// TIA Portal V17 export
// export: Created 2022-07-20T06:59:37.911436Z, ExportSetting WithDefaults, DisplayName Totally Integrated Automation Portal, DisplayVersion V17, DisplayName TIA Portal Openness, DisplayVersion V17, DisplayName TIA Portal Version Control Interface, DisplayVersion V17, DisplayName SINAMICS Startdrive Advanced, DisplayVersion V17, DisplayName SINAMICS Startdrive G130, G150, S120, S150, SINAMICS MV, S210, DisplayVersion V17, DisplayName SINAMICS Startdrive G110M, G120, G120C, G120D, G120P, G115D, DisplayVersion V17, DisplayName STEP 7 Professional, DisplayVersion V17, DisplayName STEP 7 Safety, DisplayVersion V17, DisplayName WinCC Advanced, DisplayVersion V17
FUNCTION_BLOCK "FB10010_BoolToWordAT"   // FB10010, LAD
TITLE = FB10010_BoolToWordAT
{ S7_Optimized_Access := 'TRUE' }
AUTHOR : Jonathan
FAMILY : 1001x_CONVERT
VERSION : 1.0
// Release note : 
// 1.0 - Feature developped
// stored: AutoNumber false, IsIECCheckEnabled false, IsRetainMemResEnabled false, MemoryReserve 100, SetENOAutomatically false, UDAEnableTagReadback false
   VAR_INPUT
      bool0 { ExternalAccessible := 'False'; ExternalVisible := 'False'; ExternalWritable := 'False'} : Bool;
      bool1 { ExternalAccessible := 'False'; ExternalVisible := 'False'; ExternalWritable := 'False'} : Bool;
      bool2 { ExternalAccessible := 'False'; ExternalVisible := 'False'; ExternalWritable := 'False'} : Bool;
      bool3 { ExternalAccessible := 'False'; ExternalVisible := 'False'; ExternalWritable := 'False'} : Bool;
      bool4 { ExternalAccessible := 'False'; ExternalVisible := 'False'; ExternalWritable := 'False'} : Bool;
      bool5 { ExternalAccessible := 'False'; ExternalVisible := 'False'; ExternalWritable := 'False'} : Bool;
      bool6 { ExternalAccessible := 'False'; ExternalVisible := 'False'; ExternalWritable := 'False'} : Bool;
      bool7 { ExternalAccessible := 'False'; ExternalVisible := 'False'; ExternalWritable := 'False'} : Bool;
      bool8 { ExternalAccessible := 'False'; ExternalVisible := 'False'; ExternalWritable := 'False'} : Bool;
      bool9 { ExternalAccessible := 'False'; ExternalVisible := 'False'; ExternalWritable := 'False'} : Bool;
      bool10 { ExternalAccessible := 'False'; ExternalVisible := 'False'; ExternalWritable := 'False'} : Bool;
      bool11 { ExternalAccessible := 'False'; ExternalVisible := 'False'; ExternalWritable := 'False'} : Bool;
      bool12 { ExternalAccessible := 'False'; ExternalVisible := 'False'; ExternalWritable := 'False'} : Bool;
      bool13 { ExternalAccessible := 'False'; ExternalVisible := 'False'; ExternalWritable := 'False'} : Bool;
      bool14 { ExternalAccessible := 'False'; ExternalVisible := 'False'; ExternalWritable := 'False'} : Bool;
      bool15 { ExternalAccessible := 'False'; ExternalVisible := 'False'; ExternalWritable := 'False'} : Bool;
   END_VAR
   VAR_OUTPUT
      OutWord { ExternalAccessible := 'False'; ExternalVisible := 'False'; ExternalWritable := 'False'} : Word;
   END_VAR
   VAR DB_SPECIFIC
      statOutWord : Word;
   END_VAR
   VAR
      statbools AT statOutWord : Array[0..15] of Bool;
   END_VAR
BEGIN

REGION Network 1
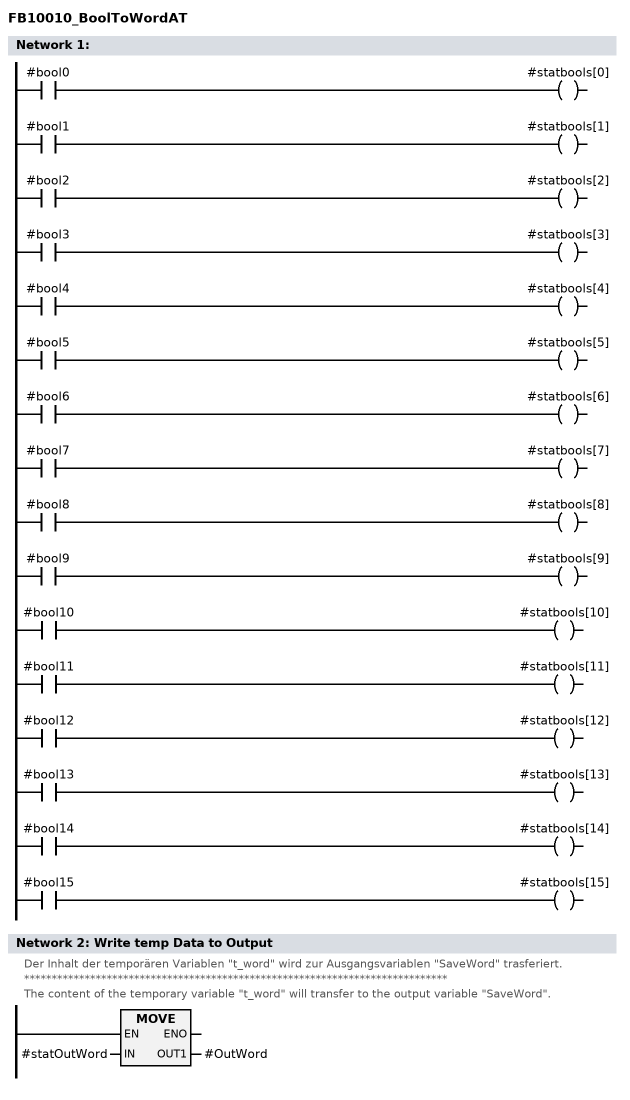
   RUNG wire#powerrail
      Contact( #bool0 )
      Coil( #statbools[0] )
   END_RUNG
   RUNG wire#powerrail
      Contact( #bool1 )
      Coil( #statbools[1] )
   END_RUNG
   RUNG wire#powerrail
      Contact( #bool2 )
      Coil( #statbools[2] )
   END_RUNG
   RUNG wire#powerrail
      Contact( #bool3 )
      Coil( #statbools[3] )
   END_RUNG
   RUNG wire#powerrail
      Contact( #bool4 )
      Coil( #statbools[4] )
   END_RUNG
   RUNG wire#powerrail
      Contact( #bool5 )
      Coil( #statbools[5] )
   END_RUNG
   RUNG wire#powerrail
      Contact( #bool6 )
      Coil( #statbools[6] )
   END_RUNG
   RUNG wire#powerrail
      Contact( #bool7 )
      Coil( #statbools[7] )
   END_RUNG
   RUNG wire#powerrail
      Contact( #bool8 )
      Coil( #statbools[8] )
   END_RUNG
   RUNG wire#powerrail
      Contact( #bool9 )
      Coil( #statbools[9] )
   END_RUNG
   RUNG wire#powerrail
      Contact( #bool10 )
      Coil( #statbools[10] )
   END_RUNG
   RUNG wire#powerrail
      Contact( #bool11 )
      Coil( #statbools[11] )
   END_RUNG
   RUNG wire#powerrail
      Contact( #bool12 )
      Coil( #statbools[12] )
   END_RUNG
   RUNG wire#powerrail
      Contact( #bool13 )
      Coil( #statbools[13] )
   END_RUNG
   RUNG wire#powerrail
      Contact( #bool14 )
      Coil( #statbools[14] )
   END_RUNG
   RUNG wire#powerrail
      Contact( #bool15 )
      Coil( #statbools[15] )
   END_RUNG
   // the same network as SCL:
   #statbools[0] := #bool0;
   #statbools[1] := #bool1;
   #statbools[2] := #bool2;
   #statbools[3] := #bool3;
   #statbools[4] := #bool4;
   #statbools[5] := #bool5;
   #statbools[6] := #bool6;
   #statbools[7] := #bool7;
   #statbools[8] := #bool8;
   #statbools[9] := #bool9;
   #statbools[10] := #bool10;
   #statbools[11] := #bool11;
   #statbools[12] := #bool12;
   #statbools[13] := #bool13;
   #statbools[14] := #bool14;
   #statbools[15] := #bool15;
END_REGION

REGION Network 2: Write temp Data to Output
   // Der Inhalt der temporären Variablen "t_word" wird zur Ausgangsvariablen "SaveWord" trasferiert.
   // *****************************************************************************
   // The content of the temporary variable "t_word" will transfer to the output variable "SaveWord".
   RUNG wire#powerrail
      { S7_GenerateENO := "TRUE" } Move(in := #statOutWord, out1 => #OutWord)
   END_RUNG
   // the same network as SCL:
   #OutWord := #statOutWord;
END_REGION
END_FUNCTION_BLOCK
